FUNCTION_BLOCK "Syntax_CaseMalformedRange"
{ S7_Optimized_Access := 'TRUE' }
VERSION : 0.1

VAR
    a        : Int := 1;
    b        : Int := 2;
    result   : Int := 0;
    flag     : Bool := TRUE;
    i        : Int := 0;
    values   : Array[0..9] of Int;
END_VAR
BEGIN
    CASE #a OF
        1...5:
            #result := 1;
        ELSE
            #result := 0;
    END_CASE;
    // EXPECT: error[syntax.invalid-case-range] SYN-CASE-003

END_FUNCTION_BLOCK
